Fanuc KAREL source: ka00143.KL

-- PROVISIONAL review KL for V770-1; original PC SHA256 33883db6d4cbf345736c60c648f4550d12fae7a8e98df36bba37ddef5d28df9e
-- Incomplete behavior may be omitted. Consult companion uncertainty JSON. Do not deploy.
PROGRAM KA00143
%NOLOCKGROUP
-- UNRESOLVED_DECL SRC type=002017
-- UNRESOLVED_DECL DST type=002018
BEGIN
  -- UNRESOLVED_PC offsets 5-19; opcodes 2E,22,9D,33,B4
  -- UNRESOLVED_PC offsets 24-42; opcodes 22,9D,33,B3,22,9D,33,B2
  -- UNRESOLVED_PC offsets 47-51; opcodes 7F
END KA00143
